FUNCTION_BLOCK TEvent_ExecutionFailed EXTENDS TEventBase IMPLEMENTS IEvent
VAR
    Message : T_MaxString;
    Handler : IEventHandler_OnExecutionFailed;
END_VAR

METHOD  CallHandler
VAR_INPUT
    HandlerBase : IEventHandlerBase;
    EventArgs   : IStreamReader;
END_VAR
VAR
    Message : T_MaxString;
END_VAR
IF __QUERYINTERFACE(HandlerBase,Handler) THEN
    Message := EventArgs.Read_STRING();
    Handler.OnExecutionFailed(Message);
END_IF
END_METHOD

METHOD  IsHandlerSupported : BOOL
VAR_INPUT
    HandlerBase : IEventHandlerBase;
END_VAR
IF __QUERYINTERFACE(HandlerBase,Handler) THEN
    IsHandlerSupported := TRUE;
END_IF
END_METHOD

END_FUNCTION_BLOCK

(* stored: Version 1.1.0.1, ProductVersion 3.1.4024.3
   POU TEvent_ExecutionFailed: Id {aba47b3c-0f39-429e-834e-e07a2e7362a1}, SpecialFunc None
   Method CallHandler: Id {e5cfdea2-747f-4019-8def-90c716dba7c3}
   Method IsHandlerSupported: Id {995a8016-bedc-46fc-a9ef-66c667f51987} *)
